TYPE Outter_coveyor :
STRUCT
	belt	: ARRAY[0..1] OF Belt;
	valve	: ARRAY[0..1] OF Valve;
	photo_sensor	: ARRAY[0..1] OF BOOL;	
END_STRUCT
END_TYPE

(* stored: Version 1.1.0.1, ProductVersion 3.1.4024.12
   DUT Outter_coveyor: Id {32b06072-052b-46a8-b5e9-bee3be0eef1f} *)
